PROGRAM PRG_MAIN
VAR

	//test: BOOL;
	//debug: INT;
	all_config_initialised: BOOL;
	FirstScan			  : BOOL:=TRUE;
	temp: INT;
	arda: INT;
	bruce: INT;
END_VAR

//Recipes
Clock();


		
IF Config.Initialised() AND bruce < 70 THEN
	bruce:=bruce+1;
ELSIF Config.Initialised() THEN   
	arda := arda+1;
	PRG_IO();
	PRG_Machine();
END_IF

FirstSCan:=FALSE;

END_PROGRAM

(* stored: Version 1.1.0.1, ProductVersion 3.1.4022.9
   POU PRG_MAIN: Id {d04c0ba0-8ee8-4b1d-b9a8-6a748878b094}, SpecialFunc None *)
